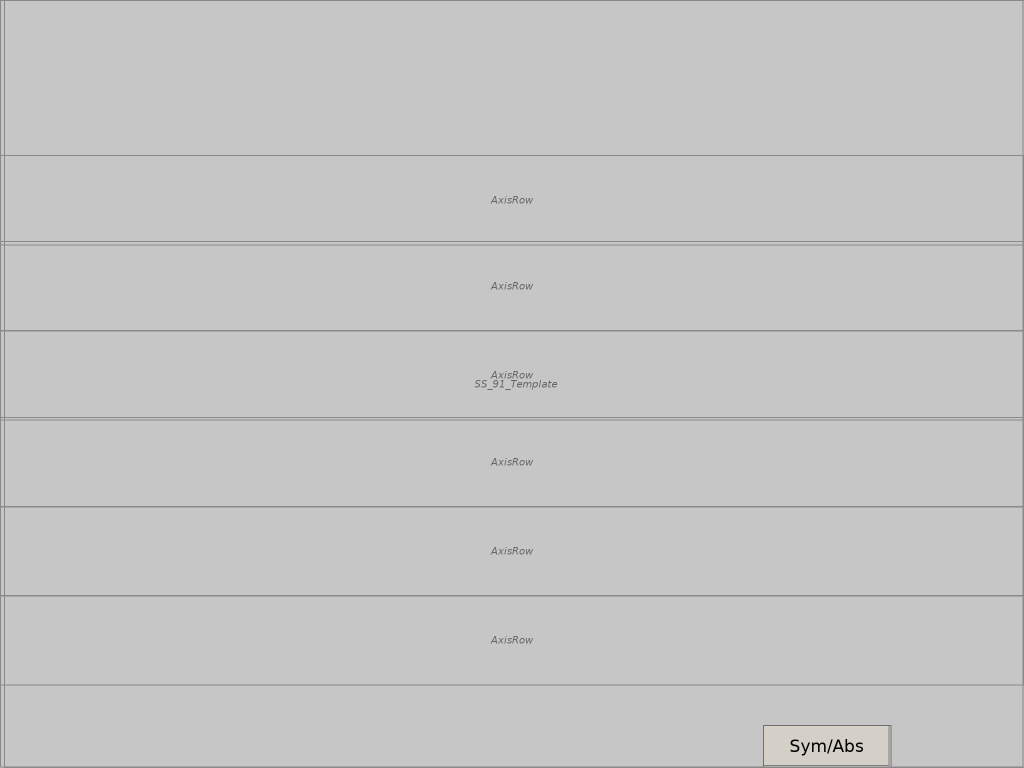
VISUALIZATION SS_13_Axis  // 1024x768
    Frame (4,0 1024x768)
        shows SS_91_Template(header := HMIData.hmiHeader)
    Frame (0,155 1024x90)
        shows AxisRow(MotionRowInstanceSingle := Axis.gAxisRows.gMotionRow1, MotionRowButtonsSingle := axis.gAxisButtons.gMotionRow1btn)
    Frame (0,241 1024x90)
        shows AxisRow(MotionRowInstanceSingle := Axis.gAxisRows.gMotionRow2, MotionRowButtonsSingle := axis.gAxisButtons.gMotionRow2btn)
    Frame (0,330 1024x90)
        shows AxisRow(MotionRowInstanceSingle := axis.gAxisRows.gMotionRow3, MotionRowButtonsSingle := axis.gAxisButtons.gMotionRow3btn)
    Frame (0,417 1024x90)
        shows AxisRow(MotionRowInstanceSingle := axis.gAxisRows.gMotionRow4, MotionRowButtonsSingle := axis.gAxisButtons.gMotionRow4btn)
    Frame (0,506 1024x90)
        shows AxisRow(MotionRowInstanceSingle := axis.gAxisRows.gMotionRow5, MotionRowButtonsSingle := axis.gAxisButtons.gMotionRow5btn)
    Frame (0,595 1024x90)
        shows AxisRow(MotionRowInstanceSingle := axis.gAxisRows.gMotionRow6, MotionRowButtonsSingle := Axis.gAxisButtons.gMotionRow6btn)
    Button (763,725 128x42), "Sym/Abs", colour toggle: HMIData.btnAbsMode
        toggle HMIData.btnAbsMode
END_VISUALIZATION

(* stored: Version 1.1.0.1, ProductVersion 3.1.4024.12
   Visu SS_13_Axis: Id {de28d113-f9c9-4f5d-a881-8399da3e9f98} *)
